{attribute 'qualified_only'}
{attribute 'strict'}
TYPE E_PneumaticAxisState :
(
    eFailSafe := 0,
    eInPosition := 1,
    eMoving := 2,
    eInterlocked := 3
) := eFailSafe;
END_TYPE

(* stored: Version 1.1.0.1
   DUT E_PneumaticAxisState: Id {6ae50a2d-0851-0276-2381-ccddacc02ce2} *)
